// TwinCAT 3 PLC project RoutinePLC
// ProgramVersion: 3.1.4024.0
// libraries:
//   Tc2_Standard, * (Beckhoff Automation GmbH)
//   Tc2_System, * (Beckhoff Automation GmbH)
//   Tc3_Module, * (Beckhoff Automation GmbH)
//   VisuDialogs, * (System)
//   VisuSymbols,3.5.10.0,System
// project tree:
//   DUTs/ Taak_1.TcDUT, Taak_2.TcDUT
//   / GlobalTextList.TcGTLO, PlcTask.TcTTO, Visualization Manager.TcVMO (not stored)
//   GVLs/ RoutineGVL.TcGVL
//   POUs/ MAIN.TcPOU, Orderverwerking_magazijn.TcPOU, POU.TcPOU, Transporteren_order.TcPOU
//   VISUs/ Orderverwerking_magazijn.TcVIS, Transporteren_order.TcVIS
// real-time tasks:
//   TASK PlcTask: cycle T#10ms, priority 20, ADS port 350

CONFIGURATION RoutinePLC
    RESOURCE PLC ON TwinCAT3
        TASK PlcTask(INTERVAL := T#10ms, PRIORITY := 20);
        PROGRAM MAIN WITH PlcTask : MAIN;
    END_RESOURCE
END_CONFIGURATION

// ---- DUTs/Taak_1.TcDUT
TYPE Taak_1 :
	(
		NieuweOrderGaragist,
		VoorraadAdministratief,
		VerzamelingArtikelen,
		OrderGeannuleerd,
		OrderVoltooid
	) := NieuweOrderGaragist;
END_TYPE

// ---- DUTs/Taak_2.TcDUT
TYPE Taak_2 :
	(
		functie,
		Inladen,
		Transport,
		Afleveren,
		Retour
	) := Inladen;
END_TYPE

// ---- GVLs/RoutineGVL.TcGVL
{attribute 'qualified_only'}
VAR_GLOBAL

END_VAR

// ---- POUs/MAIN.TcPOU
PROGRAM MAIN
VAR
END_VAR

Orderverwerking_magazijn ();
Transporteren_order();

END_PROGRAM

// ---- POUs/Orderverwerking_magazijn.TcPOU
PROGRAM Orderverwerking_magazijn
VAR
	currentState : Taak_1 := Taak_1.NieuweOrderGaragist;   
	Nieuwe_order: BOOL ;
	Order_magazijn: BOOL;
	Order_uitgeprint: BOOL;
	Timer : TON;
	WachtTijd : INT;
	Order_verzameld: BOOL; 
	Geannuleerd: BOOL;
	Order_voltooid: BOOL;
	Taak1Reset: BOOL;
	Pakfout: BOOL;
	WelOpVoorraad: BOOL;
	NietOpVoorraad: BOOL;
	Correct: BOOL;
	Incorrect: BOOL;
END_VAR

CASE currentState OF
    Taak_1.NieuweOrderGaragist:
        // Nieuwe bestelling van een garagist
        IF Nieuwe_order = TRUE THEN
            currentState := VoorraadAdministratief;
        END_IF;
		
	Taak_1.VoorraadAdministratief:
		// Controleren of de voorraad klopt (Adminastratief)
		IF WelOpVoorraad = TRUE AND Nieuwe_order = TRUE THEN
			Order_magazijn := TRUE;
			Order_uitgeprint := TRUE;
			Timer(IN:=TRUE, PT:=T#5S); 
			IF Timer.Q = TRUE THEN
				Order_verzameld := TRUE;
				Geannuleerd := FALSE;
				currentState := VerzamelingArtikelen;
				
			END_IF	
			
		ELSIF NietOpVoorraad = TRUE THEN
			currentState := OrderGeannuleerd;
		END_IF
	
		
	Taak_1.VerzamelingArtikelen:
	// Controleren of de verzamelde artikelen overeenkomen met de Orderverzamellijst
		IF Correct = TRUE THEN
			currentState := OrderVoltooid;
		ELSIF Incorrect = TRUE THEN
			currentState := OrderGeannuleerd;
		ELSIF Pakfout = TRUE THEN
			Pakfout:= TRUE;
		END_IF
		
	Taak_1.OrderVoltooid:
			Nieuwe_order := FALSE;
			WelOpVoorraad := FALSE;
			NietOpVoorraad := FALSE;
			Order_magazijn := FALSE;
			Order_uitgeprint := FALSE;
			Timer(IN:=FALSE);
			Order_verzameld := FALSE;	
			Pakfout:= FALSE;
			Order_voltooid := TRUE;		
	
	Taak_1.OrderGeannuleerd:
			Nieuwe_order := FALSE;
			WelOpVoorraad := FALSE;
			NietOpVoorraad := FALSE;
			Order_magazijn := FALSE;
			Order_uitgeprint := FALSE;
			Timer(IN:=FALSE);
			Order_verzameld := FALSE;
			Pakfout:= FALSE;
			Geannuleerd := TRUE;
		
END_CASE;
IF Taak1Reset = TRUE THEN
	currentState := Taak_1.NieuweOrderGaragist;
	Nieuwe_order := FALSE;
	WelOpVoorraad := FALSE;
	NietOpVoorraad := FALSE;
	Order_magazijn := FALSE;
	Order_uitgeprint := FALSE;
	Timer(IN:=FALSE);
	Order_verzameld := FALSE;
	Order_voltooid := FALSE;
	Geannuleerd := FALSE;
	Taak1Reset := FALSE;
	Pakfout:= FALSE;
END_IF
WachtTijd := TIME_TO_INT(timer.ET) / 1000;

END_PROGRAM

// ---- POUs/Transporteren_order.TcPOU
PROGRAM Transporteren_order
VAR
	currentState : Taak_2 := Taak_2.Functie;
	Huidige_tijd: INT := 800;
	Controleren_tijd : BOOL;
	Na10Uur: BOOL;
	Voor10Uur: BOOL;
	Wachten: BOOL;
	Inladen_krat: BOOL;
	Start_transport: BOOL;
	Timer_1 : TON;
	Timer_2 : TON;
	Locatie: BOOL;
	Afleveren : BOOL;
	
	Klant_aanwezig: BOOL;
	Klant_afwezig: BOOL;
	Afleveren_voltooid: BOOL;
	Afleveren_mislukt: BOOL;
	Retour_vestiging: BOOL;
	Taak2Reset: BOOL;

	WachtTijd_1: INT;
	WachtTijd_2: INT;
END_VAR

Controleren_tijd :=POU(Huidige_tijd);   

CASE currentState OF
	Taak_2.Functie:
		IF Controleren_tijd = TRUE THEN
			CurrentState := taak_2.inladen;
			Na10Uur := TRUE;
			Wachten := FALSE;
			Voor10Uur := FALSE;
		ELSIF Controleren_tijd = FALSE THEN
			Wachten := TRUE;
			Na10Uur := FALSE;
			Voor10Uur := TRUE;
			CurrentState := taak_2.Functie;
		END_IF
	
	Taak_2.Inladen:
		IF Controleren_tijd = TRUE THEN
			Inladen_krat := TRUE;
			Wachten := FALSE;
			CurrentState := Taak_2.Transport;
		ELSIF Controleren_tijd = FALSE THEN
			Wachten:= TRUE;
			CurrentState := taak_2.Functie;
			Inladen_krat := FALSE;
		END_IF
		
	Taak_2.Transport:
		Start_transport := TRUE; 
		Timer_1(IN:=TRUE, PT:=T#5S); 
		IF Timer_1.Q = TRUE THEN
			CurrentState := taak_2.Afleveren;
			Locatie := TRUE;
			Timer_1(IN:=FALSE);
		END_IF
	
	Taak_2.Afleveren:	
		Afleveren := TRUE;
		IF Klant_aanwezig = TRUE THEN
			Afleveren_voltooid := TRUE;
			Afleveren_mislukt := FALSE;
			Timer_2(IN:=TRUE, PT:=T#5S); 
			IF Timer_2.Q = TRUE THEN
				CurrentState := taak_2.Retour;
				Timer_2(IN:=FALSE);
			END_IF
		ELSIF Klant_afwezig = TRUE THEN
			Afleveren_mislukt := TRUE;
			Afleveren_voltooid := FALSE;
			Timer_2(IN:=TRUE, PT:=T#5S); 
			IF Timer_2.Q = TRUE THEN
				CurrentState := taak_2.Retour;
				Timer_2(IN:=FALSE);
			END_IF	
		END_IF 
	Taak_2.Retour:
		Retour_vestiging :=TRUE;
END_CASE


IF Taak2Reset = TRUE THEN
	CurrentState := taak_2.Functie;
	Huidige_tijd := 800;
	Na10Uur := FALSE;
	Wachten := FALSE;
	Voor10Uur := FALSE;
	Inladen_krat := FALSE;
	Start_transport := FALSE;
	Timer_1(IN:=FALSE);
	Timer_2(IN:=FALSE);
	Locatie := FALSE;
	Afleveren := FALSE;
	Klant_aanwezig := FALSE;
	Klant_afwezig := FALSE;
	Afleveren_voltooid := FALSE;
	Afleveren_mislukt := FALSE;
	Retour_vestiging := FALSE;
	Taak2Reset := FALSE;
END_IF
WachtTijd_1 := TIME_TO_INT(timer_1.ET) / 1000;
WachtTijd_2 := TIME_TO_INT(timer_2.ET) / 1000;

END_PROGRAM

// ---- POUs/POU.TcPOU
FUNCTION POU : BOOL
VAR_INPUT
  Huidige_tijd : INT; //Invoer van de tijd
END_VAR

IF (Huidige_tijd >= 0) AND (Huidige_tijd <= 2400) THEN
	IF Huidige_tijd >= 1000 THEN
		POU := TRUE; // Order is klaar voor transport
	ELSE
		POU := FALSE; // Order is niet klaar voor transport
	END_IF
ELSE
	POU := FALSE; //Geeft aan dat de ingevoerde tijd ongeldig is
END_IF

END_FUNCTION

// ---- GlobalTextList.TcGTLO
TEXTLIST GlobalTextList
  586 = '% Uur'
  709 = '%i'
  817 = '%I Uur'
  812 = '%i Uur'
  766 = '%s Uur'
  777 = 'Aangekomen bij vestiging'
  49 = 'Aangekomen op locatie'
  29 = 'Afleveren mislukt'
  376 = 'Afleveren voltooid'
  784 = 'c'
  223 = 'CORRECT'
  581 = 'INCORRECT (PAKFOUT)'
  3 = 'Inladen krat'
  551 = 'KLANT AANWEZIG'
  846 = 'KLANT AFWEZIG'
  543 = 'mm'
  303 = 'Na 10:00'
  886 = 'NIET OP VOORRAAD'
  648 = 'Nieuwe Order'
  625 = 'Order geannuleerd'
  809 = 'Order geanulleerd'
  791 = 'Order in behandeling'
  592 = 'Order in magazijn'
  559 = 'Order naar het magazijn'
  816 = 'Order verzameld'
  996 = 'Order verzamelen...'
  845 = 'Order Voltooid'
  725 = 'Order voltooid'
  630 = 'Orderverzamellijst geprint'
  152 = 'PAKFOUT'
  595 = 'Pakfout'
  34 = 'Reset taak'
  277 = 'Retour naar vestiging'
  289 = 'Retour naar vestiging...'
  707 = 'Rijden naar locatie...'
  930 = 'Start transport'
  820 = 'Voor 10:00'
  815 = 'Vul de huidge tijd in als volgt: (000))'
  772 = 'Vul de huidge tijd in als volgt: 0000'
  825 = 'Wachten'
  920 = 'Wat is de huige tijd? (000))'
  802 = 'Wel op voorraad'
  474 = 'WEL OP VOORRAAD'
END_TEXTLIST

// ---- VISUs/Orderverwerking_magazijn.TcVIS
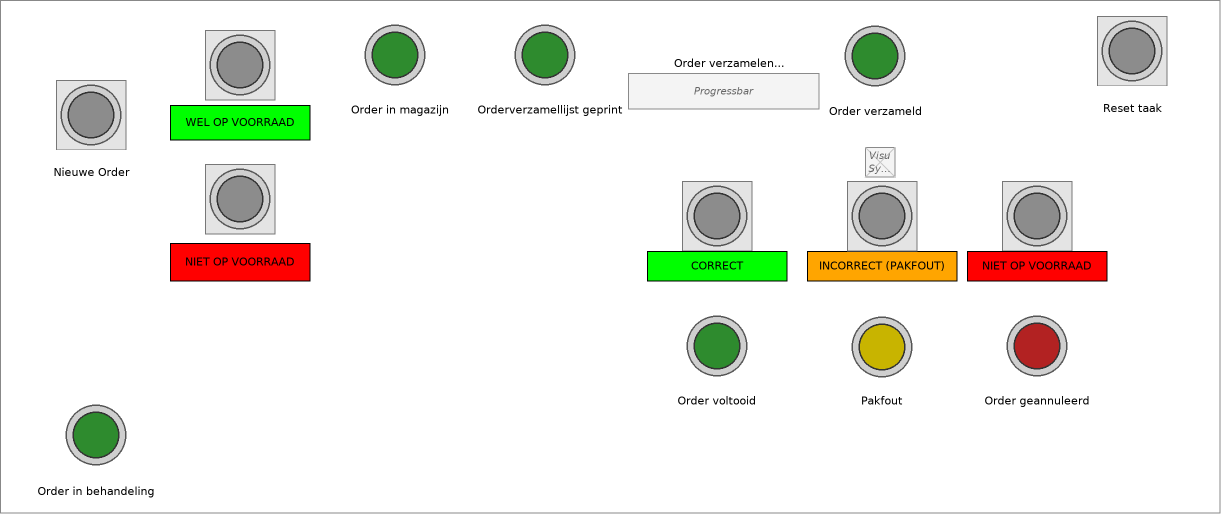
VISUALIZATION Orderverwerking_magazijn  // 1221x514
    Group (170,30 140x250)
        PushSwitch (35,0 70x70), variable: Orderverwerking_magazijn.WelOpVoorraad, behaviour: TOGGLE, style: Switch-PushSwitch-Gray
        Rectangle (0,75 140x35), "WEL OP VOORRAAD"
        PushSwitch (35,134 70x70), variable: Orderverwerking_magazijn.NietOpVoorraad, behaviour: TOGGLE, style: Switch-PushSwitch-Gray
        Rectangle (0,213 140x38), "NIET OP VOORRAAD"
    Group (30,80 120x110)
        PushSwitch (26,0 70x70), variable: Orderverwerking_magazijn.Nieuwe_order, behaviour: TOGGLE, style: Switch-PushSwitch-Gray
        Rectangle (0,70 123x45), "Nieuwe Order"
    Lamp1 (360,20 70x70), variable: Orderverwerking_magazijn.Order_magazijn, style: Lamp-Lamp1-Green
    Rectangle (340,90 120x40), "Order in magazijn"
    Lamp1 (510,20 70x70), variable: Orderverwerking_magazijn.Order_uitgeprint, style: Lamp-Lamp1-Green
    Rectangle (460,90 180x40), "Orderverzamellijst geprint"
    Group (21,400 150x114)
        Lamp1 (40,0 70x70), variable: Orderverwerking_magazijn.Nieuwe_order, style: Lamp-Lamp1-Green
        Rectangle (0,69 150x45), "Order in behandeling"
    Group (787,21 180x110)
        Lamp1 (53,0 70x70), variable: Orderverwerking_magazijn.Order_verzameld, style: Lamp-Lamp1-Green
        Rectangle (0,68 177x45), "Order verzameld"
    Group (628,41 190x70)
        Rectangle (13,0 177x45), "Order verzamelen..."
        Progressbar (0,32 191x36), variable: Orderverwerking_magazijn.WachtTijd
    Group (627,181 480x240)
        Group (335,130 150x110)
            Lamp1 (40,0 70x70), variable: Orderverwerking_magazijn.Geannuleerd, style: Lamp-Lamp1-Red
            Rectangle (0,70 150x40), "Order geannuleerd"
        Group (20,0 140x100)
            PushSwitch (35,0 70x70), variable: Orderverwerking_magazijn.Correct, behaviour: TAP, style: Switch-PushSwitch-Gray
            Rectangle (0,70 140x30), "CORRECT"
        Group (180,0 150x100)
            Rectangle (0,70 150x30), "INCORRECT (PAKFOUT)"
            PushSwitch (40,0 70x70), variable: Orderverwerking_magazijn.Pakfout, behaviour: TOGGLE, style: Switch-PushSwitch-Gray
        Group (340,0 140x100)
            PushSwitch (35,0 70x70), variable: Orderverwerking_magazijn.Incorrect, behaviour: TAP, style: Switch-PushSwitch-Gray
            Rectangle (0,70 140x30), "NIET OP VOORRAAD"
        Group (0,130 180x110)
            Lamp1 (55,0 70x70), variable: Orderverwerking_magazijn.Order_voltooid, style: Lamp-Lamp1-Green
            Rectangle (0,70 180x40), "Order voltooid"
        Group (165,131 180x109)
            Lamp1 (55,0 70x70), variable: Orderverwerking_magazijn.Pakfout, style: Lamp-Lamp1-Yellow
            Rectangle (0,69 180x40), "Pakfout"
    Group (1044,16 177x115)
        PushSwitch (53,0 70x70), variable: Orderverwerking_magazijn.Taak1Reset, behaviour: TAP, style: Switch-PushSwitch-Gray
        Rectangle (0,70 177x45), "Reset taak"
    Image (865,147 30x30), image: VisuSymbols.Symbols.ArrowBoldDown
END_VISUALIZATION

// ---- VISUs/Transporteren_order.TcVIS
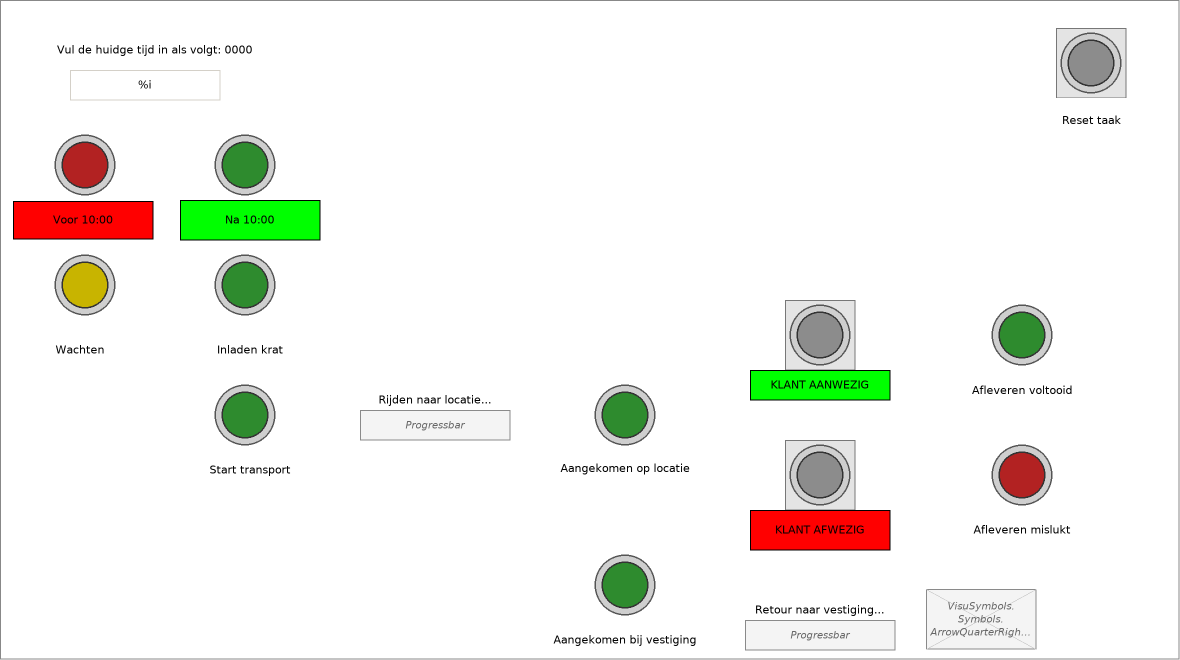
VISUALIZATION Transporteren_order  // 1180x660
    Rectangle (745,590 150x40), "Retour naar vestiging..."
    Rectangle (360,380 150x40), "Rijden naar locatie..."
    Label (40,30 230x40), "Vul de huidge tijd in als volgt: 0000"
    Textfield (70,70 150x30), "%i", text variable: Transporteren_order.Huidige_tijd
        OnMouseClick: write the text variable via Default, min 0, max 2400
    Lamp1 (50,130 70x70), variable: Transporteren_order.Voor10Uur, style: Lamp-Lamp1-Red
    Lamp1 (210,130 70x70), variable: Transporteren_order.Na10Uur, style: Lamp-Lamp1-Green
    Rectangle (13,201 140x38), "Voor 10:00"
    Rectangle (180,200 140x40), "Na 10:00"
    Lamp1 (50,250 70x70), variable: Transporteren_order.Wachten, style: Lamp-Lamp1-Yellow
    Rectangle (20,330 120x40), "Wachten"
    Lamp1 (210,250 70x70), variable: Transporteren_order.Inladen_krat, style: Lamp-Lamp1-Green
    Rectangle (190,330 120x40), "Inladen krat"
    Rectangle (190,450 120x40), "Start transport"
    Lamp1 (210,380 70x70), variable: Transporteren_order.Start_transport, style: Lamp-Lamp1-Green
    Progressbar (360,410 150x30), variable: Transporteren_order.WachtTijd_1
    Rectangle (509,446 233x45), "Aangekomen op locatie"
    Lamp1 (590,380 70x70), variable: Transporteren_order.Locatie, style: Lamp-Lamp1-Green
    PushSwitch (785,300 70x70), variable: Transporteren_order.Klant_aanwezig, behaviour: TOGGLE, style: Switch-PushSwitch-Gray
    Rectangle (750,370 140x30), "KLANT AANWEZIG"
    PushSwitch (785,440 70x70), variable: Transporteren_order.Klant_afwezig, behaviour: TOGGLE, style: Switch-PushSwitch-Gray
    Rectangle (750,510 140x40), "KLANT AFWEZIG"
    Rectangle (906,368 233x45), "Afleveren voltooid"
    Lamp1 (987,300 70x70), variable: Transporteren_order.Afleveren_voltooid, style: Lamp-Lamp1-Green
    Rectangle (907,510 230x40), "Afleveren mislukt"
    Lamp1 (987,440 70x70), variable: Transporteren_order.Afleveren_mislukt, style: Lamp-Lamp1-Red
    Image (926,589 110x60), image: VisuSymbols.Symbols.ArrowQuarterRightLeft
    Progressbar (745,620 150x30), variable: Transporteren_order.WachtTijd_2
    Lamp1 (590,550 70x70), variable: Transporteren_order.Retour_vestiging, style: Lamp-Lamp1-Green
    Rectangle (510,620 230x40), "Aangekomen bij vestiging"
    PushSwitch (1056,28 70x70), variable: Transporteren_order.Taak2Reset, behaviour: TAP, style: Switch-PushSwitch-Gray
    Rectangle (1003,98 177x45), "Reset taak"
END_VISUALIZATION
